Fanuc KAREL source: ko00072.KL

PROGRAM KO00072
%STACKSIZE=65535
%PRIORITY=65535
%NOLOCKGROUP
VAR
P1 : XYZWPREXT
P2 : XYZWPR
F : BOOLEAN
OUT : JOINTPOS9
BEGIN
F=TRUE
-- UNSAFE_SOURCE_IR line 11: CALL_RESULT MIRROR(P1, convert_xyzwpr_to_position(P2), F)
END KO00072
